{attribute 'qualified_only'}
VAR_GLOBAL
 Command : ST_Command;
 CommandCommit : UDINT;
 Status : ST_Status;
END_VAR

(* stored: Version 1.1.0.1, ProductVersion 3.1.4024.0
   GVL GVL_Hmi: Id {00000000-0000-4000-8000-000000000003} *)
